# EPICS alarm handler configuration: mps_database/bare/alarms/areas/mpln_undh_mp08.alhConfig
GROUP NULL MPLN:UNDH:MP08:1
$ALIAS MPS Link Node 143
$GUIDANCE
LTUH MPS
   Group Name: MPLN:UNDH:MP08:1
   Summary PV:  MPLN:UNDH:MP08:1:STATSUMY
$END
CHANNEL  MPLN:UNDH:MP08:1    MPLN:UNDH:MP08:1:MPS_EN_RBV		-----
CHANNEL  MPLN:UNDH:MP08:1    MPLN:UNDH:MP08:1:LC1_MODE_RBV		-----
